// TIA Portal project "Operation and manual mode lab" (V16)

(* hardware
DEVICE "S7300/ET200M station_1"  S7-300 station
   slot 0: "Rail_0"  Rail  6ES7 390-1***0-0AA0
   slot 2: "PLC_1"  CPU 315-2 DP  6ES7 315-2AH14-0AB0  V3.3
      slot 0: "MPI interface_1"  MPI
      slot 1: "DP interface_1"  DP
   slot 4: "DI 32x24VDC_1"  DI32 x 24VDC  6ES7 321-1BL00-0AA0
   slot 5: "DO 32x24VDC/0.5A_1"  DO32 x 24VDC / 0.5A  6ES7 322-1BL00-0AA0
*)

// ===== PLC "PLC_1"  CPU 315-2 DP =====

VAR_GLOBAL   // PLC tag table "Default tag table"
   "diAutoStart" AT %I0.0 : Bool;
   "diAutoStop" AT %I0.1 : Bool;
   "di1B1" AT %I2.0 : Bool;
   "di1B2" AT %I0.3 : Bool;
   "di2B1" AT %I0.4 : Bool;
   "di2B2" AT %I0.5 : Bool;
   "di3B1" AT %I0.6 : Bool;
   "di3B2" AT %I0.7 : Bool;
   "diMcStart" AT %I1.0 : Bool;
   "diMcStop" AT %I1.1 : Bool;
   "diMAN" AT %I1.2 : Bool;
   "diAUTO" AT %I1.3 : Bool;
   "diTRAN" AT %I1.4 : Bool;
   "di1A" AT %I2.1 : Bool;
   "di2A" AT %I1.6 : Bool;
   "di3A" AT %I1.7 : Bool;
   "do1Y1" AT %Q0.0 : Bool;
   "do1Y2" AT %Q0.1 : Bool;
   "do2Y1" AT %Q0.2 : Bool;
   "do2Y2" AT %Q0.3 : Bool;
   "do3Y1" AT %Q0.4 : Bool;
   "do3Y2" AT %Q0.5 : Bool;
   "doRes1" AT %Q0.6 : Bool;
   "doRes2" AT %Q0.7 : Bool;
   "doMcOn" AT %Q1.0 : Bool;
   "doMcAUTO" AT %Q1.1 : Bool;
   "doMcMan" AT %Q1.2 : Bool;
   "mMan1Y1" AT %M100.0 : Bool;
   "mMan1Y2" AT %M100.1 : Bool;
   "mMan2Y1" AT %M100.2 : Bool;
   "mMan2Y2" AT %M100.3 : Bool;
   "mMan3Y1" AT %M100.4 : Bool;
   "mMan3Y2" AT %M100.5 : Bool;
   "mAuto1Y1" AT %M101.0 : Bool;
   "mAuto1Y2" AT %M101.1 : Bool;
   "mAuto2Y1" AT %M101.2 : Bool;
   "mAuto2Y2" AT %M101.3 : Bool;
   "mAuto3Y1" AT %M101.4 : Bool;
   "mAuto3Y2" AT %M101.5 : Bool;
   "mS_Home" AT %M200.0 : Bool;
   "mS_COLeft" AT %M200.1 : Bool;
   "mAutoStart" AT %M10.0 : Bool;
   "mStart" AT %M10.1 : Bool;
   "mS_CILeft" AT %M200.2 : Bool;
   "mS_SMRight" AT %M200.3 : Bool;
   "mS_CORight" AT %M200.4 : Bool;
   "mS_CIRight" AT %M200.5 : Bool;
   "mS_SMLeft" AT %M200.6 : Bool;
END_VAR

FUNCTION "MODE" : Void   // FC10, LAD
{ S7_Optimized_Access := 'FALSE' }
VERSION : 0.1
BEGIN

REGION Network 1
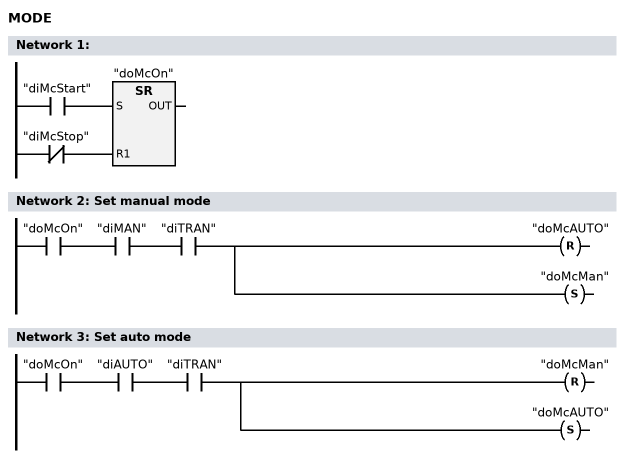
   RUNG wire#powerrail
      Contact( "diMcStart" )
      S_SR(operand := "doMcOn", r1 := wire#w1)
   END_RUNG
   RUNG wire#powerrail
      I_Contact( "diMcStop" )
   END_RUNG wire#w1
   // the same network as SCL:
   IF "diMcStart" THEN
       "doMcOn" := TRUE;   // SR flip-flop
   END_IF;
   IF NOT "diMcStop" THEN "doMcOn" := FALSE; END_IF;
END_REGION

REGION Network 2: Set manual mode
   RUNG wire#powerrail
      Contact( "doMcOn" )
      Contact( "diMAN" )
      Contact( "diTRAN" )
      wire#w1
      R_Coil( "doMcAUTO" )
   END_RUNG
   RUNG wire#w1
      S_Coil( "doMcMan" )
   END_RUNG
   // the same network as SCL:
   IF "doMcOn" AND "diMAN" AND "diTRAN" THEN
       "doMcAUTO" := FALSE;
       "doMcMan" := TRUE;
   END_IF;
END_REGION

REGION Network 3: Set auto mode
   RUNG wire#powerrail
      Contact( "doMcOn" )
      Contact( "diAUTO" )
      Contact( "diTRAN" )
      wire#w1
      R_Coil( "doMcMan" )
   END_RUNG
   RUNG wire#w1
      S_Coil( "doMcAUTO" )
   END_RUNG
   // the same network as SCL:
   IF "doMcOn" AND "diAUTO" AND "diTRAN" THEN
       "doMcMan" := FALSE;
       "doMcAUTO" := TRUE;
   END_IF;
END_REGION
END_FUNCTION

FUNCTION "MANUAL" : Void   // FC11, LAD
{ S7_Optimized_Access := 'FALSE' }
VERSION : 0.1
   VAR_TEMP   // added for the SCL form of the ladder/FBD networks
      _w1 : Bool;
   END_VAR
BEGIN

REGION Network 1: Manual Operation for CYL 1
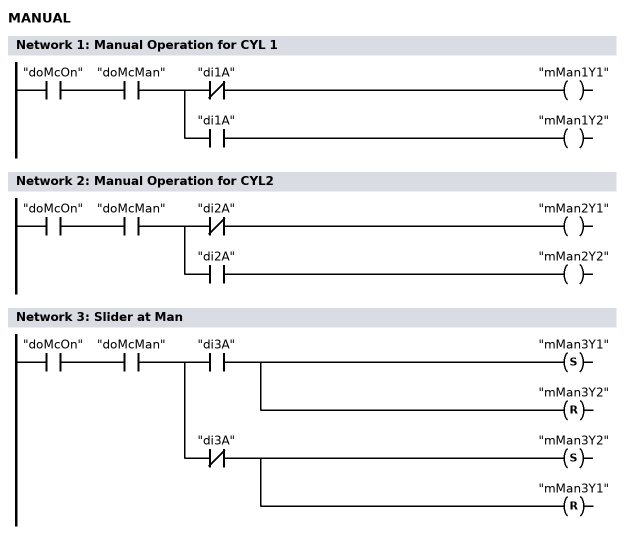
   RUNG wire#powerrail
      Contact( "doMcOn" )
      Contact( "doMcMan" )
      wire#w1
      I_Contact( "di1A" )
      Coil( "mMan1Y1" )
   END_RUNG
   RUNG wire#w1
      Contact( "di1A" )
      Coil( "mMan1Y2" )
   END_RUNG
   // the same network as SCL:
   #_w1 := "doMcOn" AND "doMcMan";
   "mMan1Y1" := #_w1 AND NOT "di1A";
   "mMan1Y2" := #_w1 AND "di1A";
END_REGION

REGION Network 2: Manual Operation for CYL2
   RUNG wire#powerrail
      Contact( "doMcOn" )
      Contact( "doMcMan" )
      wire#w1
      I_Contact( "di2A" )
      Coil( "mMan2Y1" )
   END_RUNG
   RUNG wire#w1
      Contact( "di2A" )
      Coil( "mMan2Y2" )
   END_RUNG
   // the same network as SCL:
   #_w1 := "doMcOn" AND "doMcMan";
   "mMan2Y1" := #_w1 AND NOT "di2A";
   "mMan2Y2" := #_w1 AND "di2A";
END_REGION

REGION Network 3: Slider at Man
   RUNG wire#powerrail
      Contact( "doMcOn" )
      Contact( "doMcMan" )
      wire#w1
      Contact( "di3A" )
      wire#w2
      S_Coil( "mMan3Y1" )
   END_RUNG
   RUNG wire#w2
      R_Coil( "mMan3Y2" )
   END_RUNG
   RUNG wire#w1
      I_Contact( "di3A" )
      wire#w3
      S_Coil( "mMan3Y2" )
   END_RUNG
   RUNG wire#w3
      R_Coil( "mMan3Y1" )
   END_RUNG
   // the same network as SCL:
   #_w1 := "doMcOn" AND "doMcMan";
   IF #_w1 AND "di3A" THEN
       "mMan3Y1" := TRUE;
       "mMan3Y2" := FALSE;
   END_IF;
   IF #_w1 AND NOT "di3A" THEN
       "mMan3Y2" := TRUE;
       "mMan3Y1" := FALSE;
   END_IF;
END_REGION
END_FUNCTION

FUNCTION "AUTO" : Void   // FC12, LAD
{ S7_Optimized_Access := 'FALSE' }
VERSION : 0.1
   VAR_TEMP   // added for the SCL form of the ladder/FBD networks
      _w1 : Bool;
   END_VAR
BEGIN

REGION Network 1
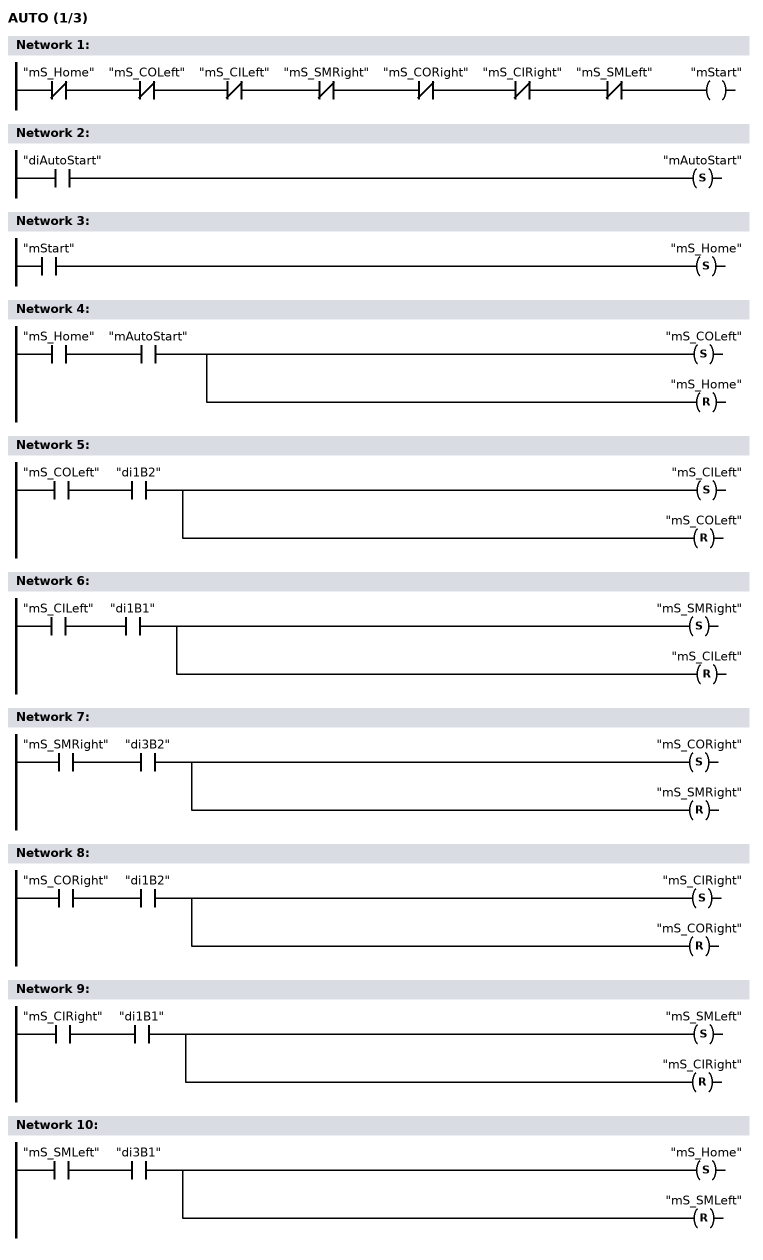
   RUNG wire#powerrail
      I_Contact( "mS_Home" )
      I_Contact( "mS_COLeft" )
      I_Contact( "mS_CILeft" )
      I_Contact( "mS_SMRight" )
      I_Contact( "mS_CORight" )
      I_Contact( "mS_CIRight" )
      I_Contact( "mS_SMLeft" )
      Coil( "mStart" )
   END_RUNG
   // the same network as SCL:
   "mStart" := NOT "mS_Home" AND NOT "mS_COLeft" AND NOT "mS_CILeft" AND NOT "mS_SMRight" AND NOT "mS_CORight" AND NOT "mS_CIRight" AND NOT "mS_SMLeft";
END_REGION

REGION Network 2
   RUNG wire#powerrail
      Contact( "diAutoStart" )
      S_Coil( "mAutoStart" )
   END_RUNG
   // the same network as SCL:
   IF "diAutoStart" THEN "mAutoStart" := TRUE; END_IF;
END_REGION

REGION Network 3
   RUNG wire#powerrail
      Contact( "mStart" )
      S_Coil( "mS_Home" )
   END_RUNG
   // the same network as SCL:
   IF "mStart" THEN "mS_Home" := TRUE; END_IF;
END_REGION

REGION Network 4
   RUNG wire#powerrail
      Contact( "mS_Home" )
      Contact( "mAutoStart" )
      wire#w1
      S_Coil( "mS_COLeft" )
   END_RUNG
   RUNG wire#w1
      R_Coil( "mS_Home" )
   END_RUNG
   // the same network as SCL:
   IF "mS_Home" AND "mAutoStart" THEN
       "mS_COLeft" := TRUE;
       "mS_Home" := FALSE;
   END_IF;
END_REGION

REGION Network 5
   RUNG wire#powerrail
      Contact( "mS_COLeft" )
      Contact( "di1B2" )
      wire#w1
      S_Coil( "mS_CILeft" )
   END_RUNG
   RUNG wire#w1
      R_Coil( "mS_COLeft" )
   END_RUNG
   // the same network as SCL:
   IF "mS_COLeft" AND "di1B2" THEN
       "mS_CILeft" := TRUE;
       "mS_COLeft" := FALSE;
   END_IF;
END_REGION

REGION Network 6
   RUNG wire#powerrail
      Contact( "mS_CILeft" )
      Contact( "di1B1" )
      wire#w1
      S_Coil( "mS_SMRight" )
   END_RUNG
   RUNG wire#w1
      R_Coil( "mS_CILeft" )
   END_RUNG
   // the same network as SCL:
   IF "mS_CILeft" AND "di1B1" THEN
       "mS_SMRight" := TRUE;
       "mS_CILeft" := FALSE;
   END_IF;
END_REGION

REGION Network 7
   RUNG wire#powerrail
      Contact( "mS_SMRight" )
      Contact( "di3B2" )
      wire#w1
      S_Coil( "mS_CORight" )
   END_RUNG
   RUNG wire#w1
      R_Coil( "mS_SMRight" )
   END_RUNG
   // the same network as SCL:
   IF "mS_SMRight" AND "di3B2" THEN
       "mS_CORight" := TRUE;
       "mS_SMRight" := FALSE;
   END_IF;
END_REGION

REGION Network 8
   RUNG wire#powerrail
      Contact( "mS_CORight" )
      Contact( "di1B2" )
      wire#w1
      S_Coil( "mS_CIRight" )
   END_RUNG
   RUNG wire#w1
      R_Coil( "mS_CORight" )
   END_RUNG
   // the same network as SCL:
   IF "mS_CORight" AND "di1B2" THEN
       "mS_CIRight" := TRUE;
       "mS_CORight" := FALSE;
   END_IF;
END_REGION

REGION Network 9
   RUNG wire#powerrail
      Contact( "mS_CIRight" )
      Contact( "di1B1" )
      wire#w1
      S_Coil( "mS_SMLeft" )
   END_RUNG
   RUNG wire#w1
      R_Coil( "mS_CIRight" )
   END_RUNG
   // the same network as SCL:
   IF "mS_CIRight" AND "di1B1" THEN
       "mS_SMLeft" := TRUE;
       "mS_CIRight" := FALSE;
   END_IF;
END_REGION

REGION Network 10
   RUNG wire#powerrail
      Contact( "mS_SMLeft" )
      Contact( "di3B1" )
      wire#w1
      S_Coil( "mS_Home" )
   END_RUNG
   RUNG wire#w1
      R_Coil( "mS_SMLeft" )
   END_RUNG
   // the same network as SCL:
   IF "mS_SMLeft" AND "di3B1" THEN
       "mS_Home" := TRUE;
       "mS_SMLeft" := FALSE;
   END_IF;
END_REGION

REGION Network 11
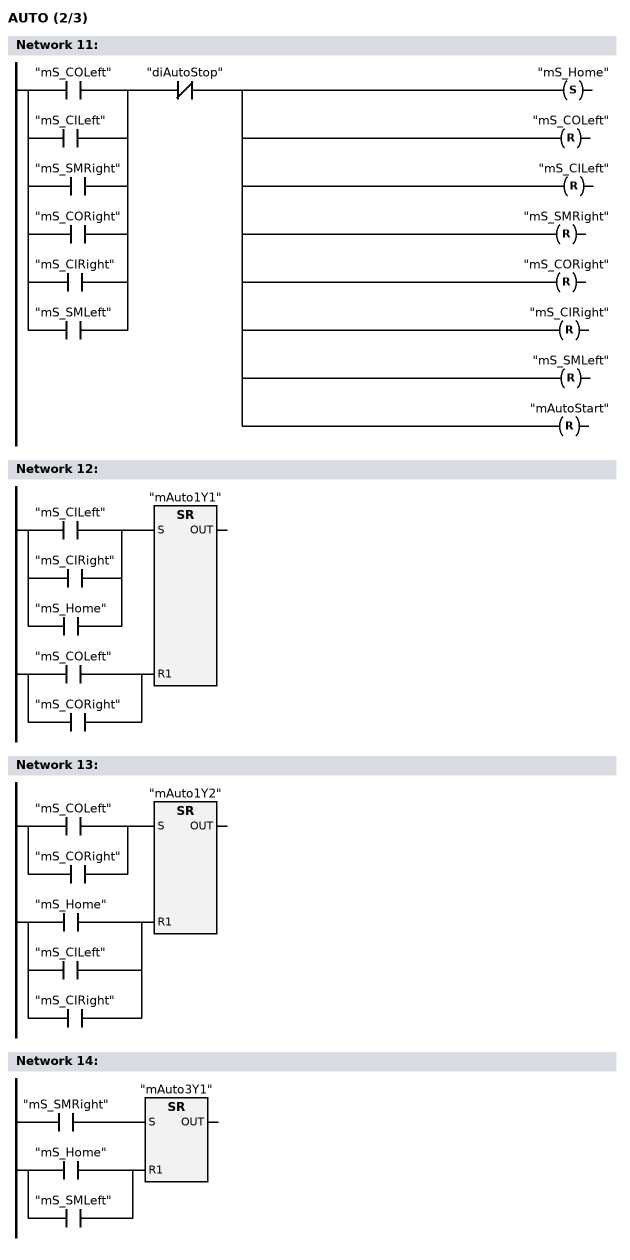
   RUNG wire#powerrail
      Contact( "mS_COLeft" )
      wire#w1
      I_Contact( "diAutoStop" )
      wire#w2
      S_Coil( "mS_Home" )
   END_RUNG
   RUNG wire#powerrail
      Contact( "mS_CILeft" )
   END_RUNG wire#w1
   RUNG wire#powerrail
      Contact( "mS_SMRight" )
   END_RUNG wire#w1
   RUNG wire#powerrail
      Contact( "mS_CORight" )
   END_RUNG wire#w1
   RUNG wire#powerrail
      Contact( "mS_CIRight" )
   END_RUNG wire#w1
   RUNG wire#powerrail
      Contact( "mS_SMLeft" )
   END_RUNG wire#w1
   RUNG wire#w2
      R_Coil( "mS_COLeft" )
   END_RUNG
   RUNG wire#w2
      R_Coil( "mS_CILeft" )
   END_RUNG
   RUNG wire#w2
      R_Coil( "mS_SMRight" )
   END_RUNG
   RUNG wire#w2
      R_Coil( "mS_CORight" )
   END_RUNG
   RUNG wire#w2
      R_Coil( "mS_CIRight" )
   END_RUNG
   RUNG wire#w2
      R_Coil( "mS_SMLeft" )
   END_RUNG
   RUNG wire#w2
      R_Coil( "mAutoStart" )
   END_RUNG
   // the same network as SCL:
   IF ("mS_COLeft" OR "mS_CILeft" OR "mS_SMRight" OR "mS_CORight" OR "mS_CIRight" OR "mS_SMLeft") AND NOT "diAutoStop" THEN
       "mS_Home" := TRUE;
   END_IF;
   #_w1 := ("mS_COLeft" OR "mS_CILeft" OR "mS_SMRight" OR "mS_CORight" OR "mS_CIRight" OR "mS_SMLeft") AND NOT "diAutoStop";
   IF #_w1 THEN
       "mS_COLeft" := FALSE;
       "mS_CILeft" := FALSE;
       "mS_SMRight" := FALSE;
       "mS_CORight" := FALSE;
       "mS_CIRight" := FALSE;
       "mS_SMLeft" := FALSE;
       "mAutoStart" := FALSE;
   END_IF;
END_REGION

REGION Network 12
   RUNG wire#powerrail
      Contact( "mS_CILeft" )
      wire#w1
      S_SR(operand := "mAuto1Y1", r1 := wire#w2)
   END_RUNG
   RUNG wire#powerrail
      Contact( "mS_CIRight" )
   END_RUNG wire#w1
   RUNG wire#powerrail
      Contact( "mS_Home" )
   END_RUNG wire#w1
   RUNG wire#powerrail
      Contact( "mS_COLeft" )
   END_RUNG wire#w2
   RUNG wire#powerrail
      Contact( "mS_CORight" )
   END_RUNG wire#w2
   // the same network as SCL:
   IF "mS_CILeft" OR "mS_CIRight" OR "mS_Home" THEN
       "mAuto1Y1" := TRUE;   // SR flip-flop
   END_IF;
   IF "mS_COLeft" OR "mS_CORight" THEN "mAuto1Y1" := FALSE; END_IF;
END_REGION

REGION Network 13
   RUNG wire#powerrail
      Contact( "mS_COLeft" )
      wire#w1
      S_SR(operand := "mAuto1Y2", r1 := wire#w2)
   END_RUNG
   RUNG wire#powerrail
      Contact( "mS_CORight" )
   END_RUNG wire#w1
   RUNG wire#powerrail
      Contact( "mS_Home" )
   END_RUNG wire#w2
   RUNG wire#powerrail
      Contact( "mS_CILeft" )
   END_RUNG wire#w2
   RUNG wire#powerrail
      Contact( "mS_CIRight" )
   END_RUNG wire#w2
   // the same network as SCL:
   IF "mS_COLeft" OR "mS_CORight" THEN
       "mAuto1Y2" := TRUE;   // SR flip-flop
   END_IF;
   IF "mS_Home" OR "mS_CILeft" OR "mS_CIRight" THEN "mAuto1Y2" := FALSE; END_IF;
END_REGION

REGION Network 14
   RUNG wire#powerrail
      Contact( "mS_SMRight" )
      S_SR(operand := "mAuto3Y1", r1 := wire#w1)
   END_RUNG
   RUNG wire#powerrail
      Contact( "mS_Home" )
   END_RUNG wire#w1
   RUNG wire#powerrail
      Contact( "mS_SMLeft" )
   END_RUNG wire#w1
   // the same network as SCL:
   IF "mS_SMRight" THEN
       "mAuto3Y1" := TRUE;   // SR flip-flop
   END_IF;
   IF "mS_Home" OR "mS_SMLeft" THEN "mAuto3Y1" := FALSE; END_IF;
END_REGION

REGION Network 15
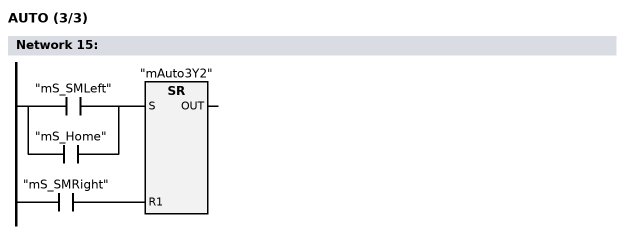
   RUNG wire#powerrail
      Contact( "mS_SMLeft" )
      wire#w1
      S_SR(operand := "mAuto3Y2", r1 := wire#w2)
   END_RUNG
   RUNG wire#powerrail
      Contact( "mS_Home" )
   END_RUNG wire#w1
   RUNG wire#powerrail
      Contact( "mS_SMRight" )
   END_RUNG wire#w2
   // the same network as SCL:
   IF "mS_SMLeft" OR "mS_Home" THEN
       "mAuto3Y2" := TRUE;   // SR flip-flop
   END_IF;
   IF "mS_SMRight" THEN "mAuto3Y2" := FALSE; END_IF;
END_REGION
END_FUNCTION

FUNCTION "OUTPUT" : Void   // FC13, LAD
{ S7_Optimized_Access := 'FALSE' }
VERSION : 0.1
BEGIN

REGION Network 1
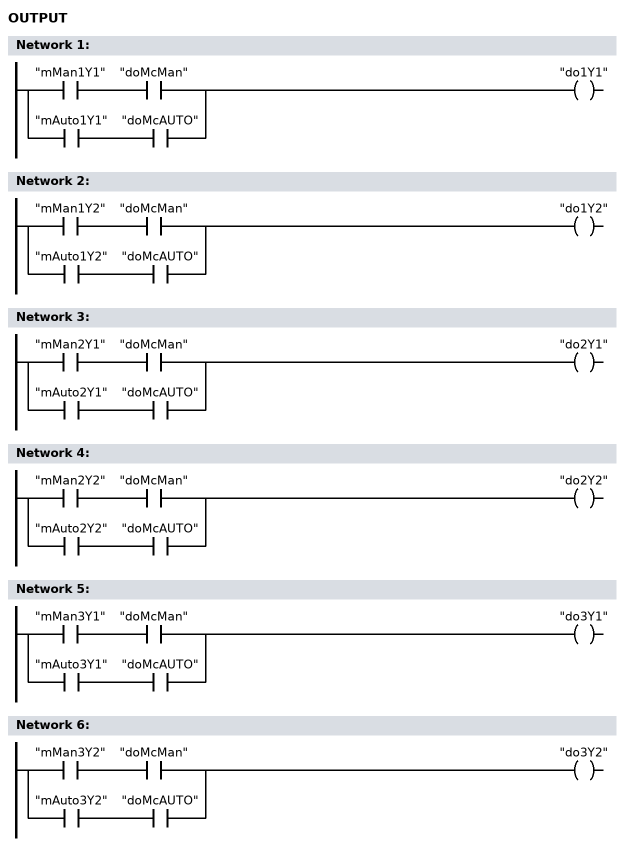
   RUNG wire#powerrail
      Contact( "mMan1Y1" )
      Contact( "doMcMan" )
      wire#w1
      Coil( "do1Y1" )
   END_RUNG
   RUNG wire#powerrail
      Contact( "mAuto1Y1" )
      Contact( "doMcAUTO" )
   END_RUNG wire#w1
   // the same network as SCL:
   "do1Y1" := ("mMan1Y1" AND "doMcMan") OR ("mAuto1Y1" AND "doMcAUTO");
END_REGION

REGION Network 2
   RUNG wire#powerrail
      Contact( "mMan1Y2" )
      Contact( "doMcMan" )
      wire#w1
      Coil( "do1Y2" )
   END_RUNG
   RUNG wire#powerrail
      Contact( "mAuto1Y2" )
      Contact( "doMcAUTO" )
   END_RUNG wire#w1
   // the same network as SCL:
   "do1Y2" := ("mMan1Y2" AND "doMcMan") OR ("mAuto1Y2" AND "doMcAUTO");
END_REGION

REGION Network 3
   RUNG wire#powerrail
      Contact( "mMan2Y1" )
      Contact( "doMcMan" )
      wire#w1
      Coil( "do2Y1" )
   END_RUNG
   RUNG wire#powerrail
      Contact( "mAuto2Y1" )
      Contact( "doMcAUTO" )
   END_RUNG wire#w1
   // the same network as SCL:
   "do2Y1" := ("mMan2Y1" AND "doMcMan") OR ("mAuto2Y1" AND "doMcAUTO");
END_REGION

REGION Network 4
   RUNG wire#powerrail
      Contact( "mMan2Y2" )
      Contact( "doMcMan" )
      wire#w1
      Coil( "do2Y2" )
   END_RUNG
   RUNG wire#powerrail
      Contact( "mAuto2Y2" )
      Contact( "doMcAUTO" )
   END_RUNG wire#w1
   // the same network as SCL:
   "do2Y2" := ("mMan2Y2" AND "doMcMan") OR ("mAuto2Y2" AND "doMcAUTO");
END_REGION

REGION Network 5
   RUNG wire#powerrail
      Contact( "mMan3Y1" )
      Contact( "doMcMan" )
      wire#w1
      Coil( "do3Y1" )
   END_RUNG
   RUNG wire#powerrail
      Contact( "mAuto3Y1" )
      Contact( "doMcAUTO" )
   END_RUNG wire#w1
   // the same network as SCL:
   "do3Y1" := ("mMan3Y1" AND "doMcMan") OR ("mAuto3Y1" AND "doMcAUTO");
END_REGION

REGION Network 6
   RUNG wire#powerrail
      Contact( "mMan3Y2" )
      Contact( "doMcMan" )
      wire#w1
      Coil( "do3Y2" )
   END_RUNG
   RUNG wire#powerrail
      Contact( "mAuto3Y2" )
      Contact( "doMcAUTO" )
   END_RUNG wire#w1
   // the same network as SCL:
   "do3Y2" := ("mMan3Y2" AND "doMcMan") OR ("mAuto3Y2" AND "doMcAUTO");
END_REGION
END_FUNCTION

ORGANIZATION_BLOCK "Main"   // OB1, LAD
TITLE = "Main Program Sweep (Cycle)"
{ S7_Optimized_Access := 'FALSE' }
VERSION : 0.1
   VAR_TEMP
      OB1_EV_CLASS : Byte;   // Bits 0-3 = 1 (Coming event), Bits 4-7 = 1 (Event class 1)
      OB1_SCAN_1 : Byte;   // 1 (Cold restart scan 1 of OB 1), 3 (Scan 2-n of OB 1)
      OB1_PRIORITY : Byte;   // Priority of OB Execution
      OB1_OB_NUMBR : Byte;   // 1 (Organization block 1, OB1)
      OB1_RESERVED_1 : Byte;   // Reserved for system
      OB1_RESERVED_2 : Byte;   // Reserved for system
      OB1_PREV_CYCLE : Int;   // Cycle time of previous OB1 scan (milliseconds)
      OB1_MIN_CYCLE : Int;   // Minimum cycle time of OB1 (milliseconds)
      OB1_MAX_CYCLE : Int;   // Maximum cycle time of OB1 (milliseconds)
      OB1_DATE_TIME : Date_And_Time;   // Date and time OB1 started
   END_VAR
BEGIN

REGION Network 1
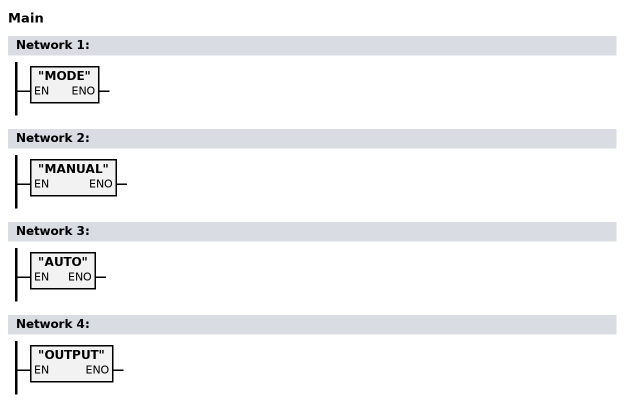
   RUNG wire#powerrail
      "MODE"()
   END_RUNG
   // the same network as SCL:
   "MODE"();
END_REGION

REGION Network 2
   RUNG wire#powerrail
      "MANUAL"()
   END_RUNG
   // the same network as SCL:
   "MANUAL"();
END_REGION

REGION Network 3
   RUNG wire#powerrail
      "AUTO"()
   END_RUNG
   // the same network as SCL:
   "AUTO"();
END_REGION

REGION Network 4
   RUNG wire#powerrail
      "OUTPUT"()
   END_RUNG
   // the same network as SCL:
   "OUTPUT"();
END_REGION
END_ORGANIZATION_BLOCK